Staubli VAL3: start.pgx

program start()
  local num l_nv
  local string l_nex
  local num l_sval
  local bool bi
  local string l_nret
begin
  call examplemenu()
end
